// TIA Portal V19 export
FUNCTION_BLOCK "FmControl"   // FB6, LAD
{ S7_Optimized_Access := 'TRUE' }
// stored: MemoryReserve 100, SetENOAutomatically false
   VAR_INPUT
      Totalise : Bool;
      "Stop & Reset Count" : Bool;
      "Stop & Preset Value" : Bool;
      "reset and totalise" : Bool;
      "Reset  & Restart" : Bool;
      "Preset and Start" : Bool;
      Hold : Bool;
   END_VAR
   VAR_OUTPUT
      FmTotaliserControl : Byte;
   END_VAR
BEGIN

REGION Network 1: The totalizer is started or continues running.
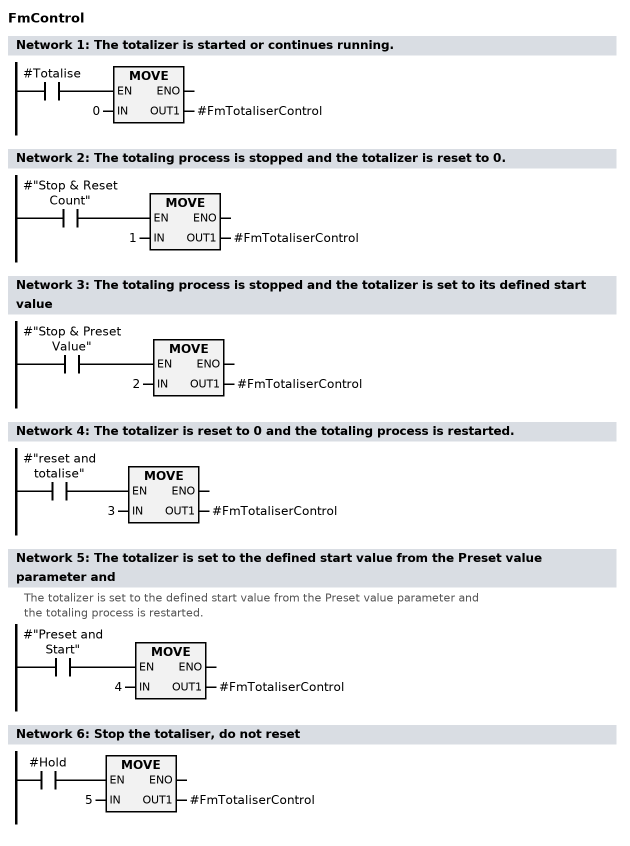
   RUNG wire#powerrail
      Contact( #Totalise )
      Move(in := 0, out1 => #FmTotaliserControl)
   END_RUNG
   // the same network as SCL:
   IF #Totalise THEN #FmTotaliserControl := 0; END_IF;
END_REGION

REGION Network 2: The totaling process is stopped and the totalizer is reset to 0.
   RUNG wire#powerrail
      Contact( #"Stop & Reset Count" )
      Move(in := 1, out1 => #FmTotaliserControl)
   END_RUNG
   // the same network as SCL:
   IF #"Stop & Reset Count" THEN #FmTotaliserControl := 1; END_IF;
END_REGION

REGION Network 3: The totaling process is stopped and the totalizer is set to its defined start value
   RUNG wire#powerrail
      Contact( #"Stop & Preset Value" )
      Move(in := 2, out1 => #FmTotaliserControl)
   END_RUNG
   // the same network as SCL:
   IF #"Stop & Preset Value" THEN #FmTotaliserControl := 2; END_IF;
END_REGION

REGION Network 4: The totalizer is reset to 0 and the totaling process is restarted.
   RUNG wire#powerrail
      Contact( #"reset and totalise" )
      Move(in := 3, out1 => #FmTotaliserControl)
   END_RUNG
   // the same network as SCL:
   IF #"reset and totalise" THEN #FmTotaliserControl := 3; END_IF;
END_REGION

REGION Network 5: The totalizer is set to the defined start value from the Preset value parameter and
   // The totalizer is set to the defined start value from the Preset value parameter and
   // the totaling process is restarted.
   RUNG wire#powerrail
      Contact( #"Preset and Start" )
      Move(in := 4, out1 => #FmTotaliserControl)
   END_RUNG
   // the same network as SCL:
   IF #"Preset and Start" THEN #FmTotaliserControl := 4; END_IF;
END_REGION

REGION Network 6: Stop the totaliser, do not reset
   RUNG wire#powerrail
      Contact( #Hold )
      Move(in := 5, out1 => #FmTotaliserControl)
   END_RUNG
   // the same network as SCL:
   IF #Hold THEN #FmTotaliserControl := 5; END_IF;
END_REGION
END_FUNCTION_BLOCK
